(* IEC 61131-3 sources: ATCMcontrol_Engineering/src/TargetBase/Libs/Modbus/eng, 48 files *)

(* ---- MODBUS_CLOSE.st ---- *)
(*[[
    UserText1= "mb_close",
    UserHelpURL= "ATCMfile:MODBUS_CLOSE.HTML",
]]*)
FUNCTION MODBUS_CLOSE : UINT
VAR_INPUT
    context : STRING; (*[context name (TCP, RTU, TCPRTU)]*)
END_VAR
INLINE {STDLIB(MODBUS_CLOSE)}
END_FUNCTION

(* ---- MODBUS_CONNECT.st ---- *)
(*[[
    UserText1= "mb_connect",
    UserHelpURL= "ATCMfile:MODBUS_CONNECT.HTML",
]]*)
FUNCTION MODBUS_CONNECT : UINT
VAR_INPUT
    context : STRING; (*[context name (TCP, RTU, TCPRTU)]*)
END_VAR
INLINE {STDLIB(MODBUS_CONNECT)}
END_FUNCTION

(* ---- MODBUS_FLUSH.st ---- *)
(*[[
    UserText1= "modbus_flush",
    UserHelpURL= "ATCMfile:MODBUS_FLUSH.HTML",
]]*)
FUNCTION MODBUS_FLUSH : UINT
VAR_INPUT
    context : STRING; (*[context name (TCP, RTU, TCPRTU)]*)
END_VAR
INLINE {STDLIB(MODBUS_FLUSH)}
END_FUNCTION

(* ---- MODBUS_FREE.st ---- *)
(*[[
    UserText1= "modbus_free",
    UserHelpURL= "ATCMfile:MODBUS_FREE.HTML",
]]*)
FUNCTION MODBUS_FREE : UINT
VAR_INPUT
    context : STRING; (*[context name (TCP, RTU, TCPRTU)]*)
END_VAR
INLINE {STDLIB(MODBUS_FREE)}
END_FUNCTION

(* ---- MODBUS_GET_BYTE_FROM_BITS.st ---- *)
(*[[
    UserText1= "mb_get_byte_from_bits",
    UserHelpURL= "ATCMfile:MODBUS_GET_BYTE_FROM_BITS.HTML",
]]*)
FUNCTION MODBUS_GET_BYTE_FROM_BITS : UINT
VAR_INPUT
	src : ARRAY[0..259] of BYTE; (*[source bit array]*)
    index : UINT; (*[index]*)
    nb_bits : UINT; (*[number of bits]*)
END_VAR
VAR_OUTPUT
	dest : BYTE; (*[byte to fill]*)
END_VAR
INLINE {STDLIB(MODBUS_GET_BYTE_FROM_BITS)}
END_FUNCTION

(* ---- MODBUS_GET_BYTE_TIMEOUT.st ---- *)
(*[[
    UserText1= "mb_get_byte_timeout",
    UserHelpURL= "ATCMfile:MODBUS_GET_BYTE_TIMEOUT.HTML",
]]*)
FUNCTION MODBUS_GET_BYTE_TIMEOUT : UINT
VAR_INPUT
    context : STRING; (*[context name (TCP, RTU, TCPRTU)]*)
END_VAR
VAR_OUTPUT
    timeout_ms : UINT; (*[timeout in milliseconds]*)
END_VAR
INLINE {STDLIB(MODBUS_GET_BYTE_TIMEOUT)}
END_FUNCTION

(* ---- MODBUS_GET_FLOAT.st ---- *)
(*[[
    UserText1= "mb_get_float",
    UserHelpURL= "ATCMfile:MODBUS_GET_FLOAT.HTML",
]]*)
FUNCTION MODBUS_GET_FLOAT : UINT
VAR_INPUT
	src : ARRAY[0..2] of UINT; (*[source bytes array]*)
END_VAR
VAR_OUTPUT
	value : REAL; (*[float value]*)
END_VAR
INLINE {STDLIB(MODBUS_GET_FLOAT)}
END_FUNCTION

(* ---- MODBUS_GET_FLOAT_BADC.st ---- *)
(*[[
    UserText1= "mb_get_float_badc",
    UserHelpURL= "ATCMfile:MODBUS_GET_FLOAT_BADC.HTML",
]]*)
FUNCTION MODBUS_GET_FLOAT_BADC : UINT
VAR_INPUT
	src : ARRAY[0..2] of UINT; (*[source bytes array]*)
END_VAR
VAR_OUTPUT
	value : REAL; (*[float value]*)
END_VAR
INLINE {STDLIB(MODBUS_GET_FLOAT_BADC)}
END_FUNCTION

(* ---- MODBUS_GET_FLOAT_CDAB.st ---- *)
(*[[
    UserText1= "mb_get_float_cdab",
    UserHelpURL= "ATCMfile:MODBUS_GET_FLOAT_CDAB.HTML",
]]*)
FUNCTION MODBUS_GET_FLOAT_CDAB : UINT
VAR_INPUT
	src : ARRAY[0..2] of UINT; (*[source bytes array]*)
END_VAR
VAR_OUTPUT
	value : REAL; (*[float value]*)
END_VAR
INLINE {STDLIB(MODBUS_GET_FLOAT_CDAB)}
END_FUNCTION

(* ---- MODBUS_GET_FLOAT_DCBA.st ---- *)
(*[[
    UserText1= "mb_get_float_dcba",
    UserHelpURL= "ATCMfile:MODBUS_GET_FLOAT_DCBA.HTML",
]]*)
FUNCTION MODBUS_GET_FLOAT_DCBA : UINT
VAR_INPUT
	src : ARRAY[0..2] of UINT; (*[source bytes array]*)
END_VAR
VAR_OUTPUT
	value : REAL; (*[float value]*)
END_VAR
INLINE {STDLIB(MODBUS_GET_FLOAT_DCBA)}
END_FUNCTION

(* ---- MODBUS_GET_HEADER_LENGTH.st ---- *)
(*[[
    UserText1= "mb_get_header_length",
    UserHelpURL= "ATCMfile:MODBUS_GET_HEADER_LENGTH.HTML",
]]*)
FUNCTION MODBUS_GET_HEADER_LENGTH : UINT
VAR_INPUT
    context : STRING; (*[context name (TCP, RTU, TCPRTU)]*)
END_VAR
INLINE {STDLIB(MODBUS_GET_HEADER_LENGTH)}
END_FUNCTION

(* ---- MODBUS_GET_RESPONSE_TIMEOUT.st ---- *)
(*[[
    UserText1= "mb_get_response_timeout",
    UserHelpURL= "ATCMfile:MODBUS_GET_RESPONSE_TIMEOUT.HTML",
]]*)
FUNCTION MODBUS_GET_RESPONSE_TIMEOUT : UINT
VAR_INPUT
    context : STRING; (*[context name (TCP, RTU, TCPRTU)]*)
END_VAR
VAR_OUTPUT
    timeout_ms : UINT; (*[timeout in milliseconds]*)
END_VAR
INLINE {STDLIB(MODBUS_GET_RESPONSE_TIMEOUT)}
END_FUNCTION

(* ---- MODBUS_MASK_WRITE_REGISTER.st ---- *)
(*[[
    UserText1= "mb_mask_write_register",
    UserHelpURL= "ATCMfile:MODBUS_MASK_WRITE_REGISTER.HTML",
]]*)
FUNCTION MODBUS_MASK_WRITE_REGISTER : UINT
VAR_INPUT
    context : STRING; (*[context name (TCP, RTU, TCPRTU)]*)
    addr : UINT; (*[address from start to read]*)
    and_mask : UINT; (*[AND mask]*)
    or_mask : UINT; (*[OR mask]*)
END_VAR
INLINE {STDLIB(MODBUS_MASK_WRITE_REGISTER)}
END_FUNCTION

(* ---- MODBUS_NEW_RTU.st ---- *)
(*[[
    UserText1= "mb_new_rtu",
    UserHelpURL= "ATCMfile:MODBUS_NEW_RTU.HTML",
]]*)
FUNCTION MODBUS_NEW_RTU : UINT
VAR_INPUT
    device : STRING; (*[device to connect]*)
    baud : UINT; (*[baud rate]*)
    parity : STRING; (*[parity bit]*)
    data_bit : UINT; (*[nb of data bit]*)
    stop_bit : UINT; (*[nb of stop bit]*)
END_VAR
INLINE {STDLIB(MODBUS_NEW_RTU)}
END_FUNCTION

(* ---- MODBUS_NEW_TCP.st ---- *)
(*[[
    UserText1= "mb_new_tcp",
    UserHelpURL= "ATCMfile:MODBUS_NEW_TCP.HTML",
]]*)
FUNCTION MODBUS_NEW_TCP : UINT
VAR_INPUT
    ip_address : STRING; (*[ip address to connect]*)
    port : UINT; (*[port to connect]*)
END_VAR
INLINE {STDLIB(MODBUS_NEW_TCP)}
END_FUNCTION

(* ---- MODBUS_NEW_TCP_PI.st ---- *)
(*[[
    UserText1= "mb_new_tcp_pi",
    UserHelpURL= "ATCMfile:MODBUS_NEW_TCP_PI.HTML",
]]*)
FUNCTION MODBUS_NEW_TCP_PI : UINT
VAR_INPUT
    node : STRING; (*[node name]*)
    service : STRING; (*[service name]*)
END_VAR
INLINE {STDLIB(MODBUS_NEW_TCP_PI)}
END_FUNCTION

(* ---- MODBUS_NEW_TCPRTU.st ---- *)
(*[[
    UserText1= "mb_new_tcprtu",
    UserHelpURL= "ATCMfile:MODBUS_NEW_TCPRTU.HTML",
]]*)
FUNCTION MODBUS_NEW_TCPRTU : UINT
VAR_INPUT
    ip_address : STRING; (*[ip address to connect]*)
    port : UINT; (*[port to connect]*)
END_VAR
INLINE {STDLIB(MODBUS_NEW_TCPRTU)}
END_FUNCTION

(* ---- MODBUS_READ_BITS.st ---- *)
(*[[
    UserText1= "mb_read_bits",
    UserHelpURL= "ATCMfile:MODBUS_READ_BITS.HTML",
]]*)
FUNCTION MODBUS_READ_BITS : UINT
VAR_INPUT
    context : STRING; (*[context name (TCP, RTU, TCPRTU)]*)
    addr : UINT; (*[address from start to read]*)
    nb_bits : UINT; (*[number of bits]*)
END_VAR
VAR_OUTPUT
	data : ARRAY[0..259] of BYTE; (*[bits read]*)
END_VAR
INLINE {STDLIB(MODBUS_READ_BITS)}
END_FUNCTION

(* ---- MODBUS_READ_INPUT_BITS.st ---- *)
(*[[
    UserText1= "mb_read_input_bits",
    UserHelpURL= "ATCMfile:MODBUS_READ_BITS.HTML",
]]*)
FUNCTION MODBUS_READ_INPUT_BITS : UINT
VAR_INPUT
    context : STRING; (*[context name (TCP, RTU, TCPRTU)]*)
    addr : UINT; (*[address from start to read]*)
    nb_bits : UINT; (*[number of bits to read]*)
END_VAR
VAR_OUTPUT
	data : ARRAY[0..259] of BOOL; (*[bits read]*)
END_VAR
INLINE {STDLIB(MODBUS_READ_INPUT_BITS)}
END_FUNCTION

(* ---- MODBUS_READ_INPUT_REGISTERS.st ---- *)
(*[[
    UserText1= "mb_read_input_registers",
    UserHelpURL= "ATCMfile:MODBUS_READ_INPUT_REGISTERS.HTML",
]]*)
FUNCTION MODBUS_READ_INPUT_REGISTERS : UINT
VAR_INPUT
    context : STRING; (*[context name (TCP, RTU, TCPRTU)]*)
    addr : UINT; (*[address from start to read]*)
    nb_regs : UINT; (*[number of register to read]*)
END_VAR
VAR_OUTPUT
	data : ARRAY[0..259] of UINT; (*[registers read]*)
END_VAR
INLINE {STDLIB(MODBUS_READ_INPUT_REGISTERS)}
END_FUNCTION

(* ---- MODBUS_READ_REGISTERS.st ---- *)
(*[[
    UserHelpURL= "ATCMfile:MODBUS_READ_REGISTERS.HTML",
    UserText1= "mb_read_registers",
]]*)
FUNCTION MODBUS_READ_REGISTERS : UINT
VAR_INPUT
    context : STRING; (*[context name (TCP, RTU, TCPRTU)]*)
    addr : UINT; (*[address from start to read]*)
    nb_regs : UINT; (*[number of register to read]*)
END_VAR
VAR_OUTPUT
	data : ARRAY[0..259] of UINT; (*[registers read]*)
END_VAR
INLINE {STDLIB(MODBUS_READ_REGISTERS)}
END_FUNCTION

(* ---- MODBUS_REPORT_SLAVE_ID.st ---- *)
(*[[
    UserText1= "mb_report_slave_id",
    UserHelpURL= "ATCMfile:MODBUS_REPORT_SLAVE_ID.HTML",
]]*)
FUNCTION MODBUS_REPORT_SLAVE_ID : UINT
VAR_INPUT
    context : STRING; (*[context name (TCP, RTU, TCPRTU)]*)
END_VAR
VAR_OUTPUT
	dest : ARRAY[0..259] of BYTE; (*[slave id report]*)
END_VAR
INLINE {STDLIB(MODBUS_REPORT_SLAVE_ID)}
END_FUNCTION

(* ---- MODBUS_RTU_GET_RTS.st ---- *)
(*[[
    UserText1= "mb_rtu_get_rts",
    UserHelpURL= "ATCMfile:MODBUS_RTU_GET_RTS.HTML",
]]*)
FUNCTION MODBUS_RTU_GET_RTS : UINT
VAR_OUTPUT
    rts : UINT; (*[rtu rts]*)
END_VAR
INLINE {STDLIB(MODBUS_RTU_GET_RTS)}
END_FUNCTION

(* ---- MODBUS_RTU_GET_SERIAL_MODE.st ---- *)
(*[[
    UserText1= "mb_rtu_get_serial_mode",
    UserHelpURL= "ATCMfile:MODBUS_RTU_GET_SERIAL_MODE.HTML",
]]*)
FUNCTION MODBUS_RTU_GET_SERIAL_MODE : UINT
VAR_OUTPUT
    mode : UINT; (*[mode]*)
END_VAR
INLINE {STDLIB(MODBUS_RTU_GET_SERIAL_MODE)}
END_FUNCTION

(* ---- MODBUS_RTU_SET_RTS.st ---- *)
(*[[
    UserText1= "mb_rtu_set_rts",
    UserHelpURL= "ATCMfile:MODBUS_RTU_SET_RTS.HTML",
]]*)
FUNCTION MODBUS_RTU_SET_RTS : UINT
VAR_INPUT
    rts : UINT; (*[rtu rts]*)
END_VAR
INLINE {STDLIB(MODBUS_RTU_SET_RTS)}
END_FUNCTION

(* ---- MODBUS_RTU_SET_SERIAL_MODE.st ---- *)
(*[[
    UserText1= "mb_rtu_set_serial_mode",
    UserHelpURL= "ATCMfile:MODBUS_RTU_SET_SERIAL_MODE.HTML",
]]*)
FUNCTION MODBUS_RTU_SET_SERIAL_MODE : UINT
VAR_INPUT
    mode : UINT; (*[mode]*)
END_VAR
INLINE {STDLIB(MODBUS_RTU_SET_SERIAL_MODE)}
END_FUNCTION

(* ---- MODBUS_SET_BITS_FROM_BYTE.st ---- *)
(*[[
    UserText1= "mb_set_bits_from_byte",
    UserHelpURL= "ATCMfile:MODBUS_SET_BITS_FROM_BYTE.HTML",
]]*)
FUNCTION MODBUS_SET_BITS_FROM_BYTE : UINT
VAR_INPUT
    index : UINT; (*[index]*)
    value : BYTE; (*[source byte]*)
END_VAR
VAR_OUTPUT
	dest : ARRAY[0..259] of BYTE; (*[bits array to fill]*)
END_VAR
INLINE {STDLIB(MODBUS_SET_BITS_FROM_BYTE)}
END_FUNCTION

(* ---- MODBUS_SET_BITS_FROM_BYTES.st ---- *)
(*[[
    UserText1= "mb_set_bits_from_bytes",
    UserHelpURL= "ATCMfile:MODBUS_SET_BITS_FROM_BYTES.HTML",
]]*)
FUNCTION MODBUS_SET_BITS_FROM_BYTES : UINT
VAR_INPUT
	tab_byte : ARRAY[0..259] of BYTE; (*[source bytes array]*)
    index : UINT; (*[index]*)
    nb_bits : UINT; (*[number of bits]*)
END_VAR
VAR_OUTPUT
	dest : ARRAY[0..259] of BYTE; (*[bits array to fill]*)
END_VAR
INLINE {STDLIB(MODBUS_SET_BITS_FROM_BYTES)}
END_FUNCTION

(* ---- MODBUS_SET_BITS_FROM_BYTES_PARAM.st ---- *)
(*[[
    UserText1= "mb_set_bits_from_bytes",
    UserHelpURL= "ATCMfile:MODBUS_SET_BITS_FROM_BYTES_PARAM.HTML",
]]*)
FUNCTION MODBUS_SET_BITS_FROM_BYTES_PARAM : UINT
VAR_INPUT
	tab_byte : ARRAY[0..260] of UINT; (*[source bytes array]*)
    index : UINT; (*[index]*)
    nb_bits : UINT; (*[number of bits]*)
END_VAR
VAR_OUTPUT
	dest : ARRAY[0..260] of UINT; (*[bits array to fill]*)
END_VAR
INLINE {STDLIB(MODBUS_SET_BITS_FROM_BYTES_PARAM)}
END_FUNCTION

(* ---- MODBUS_SET_BYTE_TIMEOUT.st ---- *)
(*[[
    UserText1= "mb_set_byte_timeout",
    UserHelpURL= "ATCMfile:MODBUS_SET_BYTE_TIMEOUT.HTML",
]]*)
FUNCTION MODBUS_SET_BYTE_TIMEOUT : UINT
VAR_INPUT
    context : STRING; (*[context name (TCP, RTU, TCPRTU)]*)
    timeout_ms : UINT; (*[timeout in milliseconds]*)
END_VAR
INLINE {STDLIB(MODBUS_SET_BYTE_TIMEOUT)}
END_FUNCTION

(* ---- MODBUS_SET_ERROR_RECOVERY.st ---- *)
(*[[
  UserText1= "mb_set_error_recovery",
    UserHelpURL= "ATCMfile:MODBUS_SET_ERROR_RECOVERY.HTML",
]]*)
FUNCTION MODBUS_SET_ERROR_RECOVERY

VAR_INPUT
    context : STRING; (*[context name (TCP, RTU, TCPRTU)]*)
    recovery_mode : UINT; (*[recovery mode: 0 - NONE , 1 - LINK, 2 - PROTOCOL]*)
END_VAR
INLINE {STDLIB(MODBUS_SET_ERROR_RECOVERY)}
END_FUNCTION

(* ---- MODBUS_SET_FLOAT.st ---- *)
(*[[
    UserText1= "mb_set_float",
    UserHelpURL= "ATCMfile:MODBUS_SET_FLOAT.HTML",
]]*)
FUNCTION MODBUS_SET_FLOAT : UINT
VAR_INPUT
	dest : ARRAY[0..2] of UINT; (*[source bytes array]*)
	value : REAL; (*[float value]*)
END_VAR
INLINE {STDLIB(MODBUS_SET_FLOAT)}
END_FUNCTION

(* ---- MODBUS_SET_FLOAT_BADC.st ---- *)
(*[[
    UserText1= "mb_set_float_badc",
    UserHelpURL= "ATCMfile:MODBUS_SET_FLOAT_BADC.HTML",
]]*)
FUNCTION MODBUS_SET_FLOAT_BADC : UINT
VAR_INPUT
	dest : ARRAY[0..2] of UINT; (*[source bytes array]*)
	value : REAL; (*[float value]*)
END_VAR
INLINE {STDLIB(MODBUS_SET_FLOAT_BADC)}END_FUNCTION

(* ---- MODBUS_SET_FLOAT_CDAB.st ---- *)
(*[[
    UserText1= "mb_set_float_cdab",
    UserHelpURL= "ATCMfile:MODBUS_SET_FLOAT_CDAB.HTML",
]]*)
FUNCTION MODBUS_SET_FLOAT_CDAB : UINT
VAR_INPUT
	dest : ARRAY[0..2] of UINT; (*[source bytes array]*)
	value : REAL; (*[float value]*)
END_VAR
INLINE {STDLIB(MODBUS_SET_FLOAT_CDAB)}END_FUNCTION

(* ---- MODBUS_SET_FLOAT_DCBA.st ---- *)
(*[[
    UserText1= "mb_set_float_dcba",
    UserHelpURL= "ATCMfile:MODBUS_SET_FLOAT_DCBA.HTML",
]]*)
FUNCTION MODBUS_SET_FLOAT_DCBA : UINT
VAR_INPUT
	dest : ARRAY[0..2] of UINT; (*[source bytes array]*)
	value : REAL; (*[float value]*)
END_VAR
INLINE {STDLIB(MODBUS_SET_FLOAT_DCBA)}END_FUNCTION

(* ---- MODBUS_SET_RESPONSE_TIMEOUT.st ---- *)
(*[[
    UserText1= "mb_set_response_timeout",
    UserHelpURL= "ATCMfile:MODBUS_SET_RESPONSE_TIMEOUT.HTML",
]]*)
FUNCTION MODBUS_SET_RESPONSE_TIMEOUT : UINT
VAR_INPUT
    context : STRING; (*[context name (TCP, RTU, TCPRTU)]*)
    timeout_ms : UINT; (*[timeout in milliseconds]*)
END_VAR
INLINE {STDLIB(MODBUS_SET_RESPONSE_TIMEOUT)}
END_FUNCTION

(* ---- MODBUS_SET_SLAVE.st ---- *)
(*[[
    UserText1= "mb_set_slave",
    UserHelpURL= "ATCMfile:MODBUS_SET_SLAVE.HTML",
]]*)
FUNCTION MODBUS_SET_SLAVE : UINT
VAR_INPUT
    context : STRING; (*[context name (TCP, RTU, TCPRTU)]*)
    slave : BYTE; (*[salve id]*)
END_VAR
INLINE {STDLIB(MODBUS_SET_SLAVE)}
END_FUNCTION

(* ---- MODBUS_TCP_ACCEPT.st ---- *)
(*[[
    UserText1= "mb_tcp_accept",
    UserHelpURL= "ATCMfile:MODBUS_TCP_ACCEPT.HTML",
]]*)
FUNCTION MODBUS_TCP_ACCEPT : UINT
INLINE {STDLIB(MODBUS_TCP_ACCEPT)}
END_FUNCTION

(* ---- MODBUS_TCP_LISTEN.st ---- *)
(*[[
    UserText1= "mb_tcp_listen",
    UserHelpURL= "ATCMfile:MODBUS_TCP_LISTEN.HTML",
]]*)
FUNCTION MODBUS_TCP_LISTEN : UINT
INLINE {STDLIB(MODBUS_TCP_LISTEN)}
END_FUNCTION

(* ---- MODBUS_TCP_PI_ACCEPT.st ---- *)
(*[[
    UserHelpURL= "ATCMfile:MODBUS_TCP_PI_ACCEPT.HTML",
    UserText1= "mb_tcp_pi_accept",
]]*)
FUNCTION MODBUS_TCP_PI_ACCEPT : UINT
INLINE {STDLIB(MODBUS_TCP_PI_ACCEPT)}
END_FUNCTION

(* ---- MODBUS_TCP_PI_LISTEN.st ---- *)
(*[[
    UserText1= "mb_tcp_pi_listen",
    UserHelpURL= "ATCMfile:MODBUS_TCP_PI_LISTEN.HTML",
]]*)
FUNCTION MODBUS_TCP_PI_LISTEN : UINT
INLINE {STDLIB(MODBUS_TCP_PI_LISTEN)}
END_FUNCTION

(* ---- MODBUS_TCPRTU_ACCEPT.st ---- *)
(*[[
    UserText1= "mb_tcprtu_accept",
    UserHelpURL= "ATCMfile:MODBUS_TCPRTU_ACCEPT.HTML",
]]*)
FUNCTION MODBUS_TCPRTU_ACCEPT : UINT
INLINE {STDLIB(MODBUS_TCPRTU_ACCEPT)}
END_FUNCTION

(* ---- MODBUS_TCPRTU_LISTEN.st ---- *)
(*[[
    UserText1= "mb_tcprtu_listen",
    UserHelpURL= "ATCMfile:MODBUS_TCPRTU_LISTEN.HTML",
]]*)
FUNCTION MODBUS_TCPRTU_LISTEN : UINT
INLINE {STDLIB(MODBUS_TCPRTU_LISTEN)}
END_FUNCTION

(* ---- MODBUS_WRITE_AND_READ_REGISTERS.st ---- *)
(*[[
    UserText1= "mb_write_and_read_registers",
    UserHelpURL= "ATCMfile:MODBUS_WRITE_AND_READ_REGISTERS.HTML",
]]*)
FUNCTION MODBUS_WRITE_AND_READ_REGISTERS : UINT
VAR_INPUT
    context : STRING; (*[context name (TCP, RTU, TCPRTU)]*)
    write_addr : DINT; (*[address from start to write]*)
	src : ARRAY[0..259] of UINT; (*[bits to write]*)
    write_nb : UINT; (*[number of register to write]*)
    read_addr : DINT; (*[address from start to read]*)
    read_nb : UINT; (*[number of register to read]*)
END_VAR
VAR_OUTPUT
	dest : ARRAY[0..259] of UINT; (*[bits to write]*)
END_VAR
INLINE {STDLIB(MODBUS_WRITE_AND_READ_REGISTERS)}
END_FUNCTION

(* ---- MODBUS_WRITE_BIT.st ---- *)
(*[[
    UserText1= "mb_write_bit",
    UserHelpURL= "ATCMfile:MODBUS_WRITE_BIT.HTML",
]]*)
FUNCTION MODBUS_WRITE_BIT : UINT
VAR_INPUT
    context : STRING; (*[context name (TCP, RTU, TCPRTU)]*)
    addr : UINT; (*[address from start to read]*)
    status : INT; (*[status to set to the bit]*)
END_VAR
INLINE {STDLIB(MODBUS_WRITE_BIT)}
END_FUNCTION

(* ---- MODBUS_WRITE_BITS.st ---- *)
(*[[
    UserText1= "mb_write_bits",
    UserHelpURL= "ATCMfile:MODBUS_WRITE_BITS.HTML",
]]*)
FUNCTION MODBUS_WRITE_BITS : UINT
VAR_INPUT
    context : STRING; (*[context name (TCP, RTU, TCPRTU)]*)
    addr : UINT; (*[address from start to read]*)
    nb_bits : UINT; (*[number of bits]*)
	data : ARRAY[0..259] of BYTE; (*[bits array write]*)
END_VAR
INLINE {STDLIB(MODBUS_WRITE_BITS)}
END_FUNCTION

(* ---- MODBUS_WRITE_REGISTER.st ---- *)
(*[[
    UserText1= "mb_write_register",
    UserHelpURL= "ATCMfile:MODBUS_WRITE_REGISTER.HTML",
]]*)
FUNCTION MODBUS_WRITE_REGISTER : UINT
VAR_INPUT
    context : STRING; (*[context name (TCP, RTU, TCPRTU)]*)
    addr : UINT; (*[address from start to read]*)
	data : UINT; (*[register to write]*)
END_VAR
INLINE {STDLIB(MODBUS_WRITE_REGISTER)}
END_FUNCTION

(* ---- MODBUS_WRITE_REGISTERS.st ---- *)
(*[[
    UserText1= "mb_write_registers",
    UserHelpURL= "ATCMfile:MODBUS_WRITE_REGISTERS.HTML",
]]*)
FUNCTION MODBUS_WRITE_REGISTERS : UINT
VAR_INPUT
    context : STRING; (*[context name (TCP, RTU, TCPRTU)]*)
    addr : UINT; (*[address from start to read]*)
    status : INT; (*[status to set to the bit]*)
	data : ARRAY[0..259] of UINT; (*[register to write]*)
END_VAR
INLINE {STDLIB(MODBUS_WRITE_REGISTERS)}
END_FUNCTION
